FUNCTION_BLOCK StartStopEvents (* Basic Function Block Type *)
  (* Standard: 61499-2 *)
  (* Version 0.0, 18/05/2022, Admin, Schneider Electric, Template *)
  PACKAGE Main;
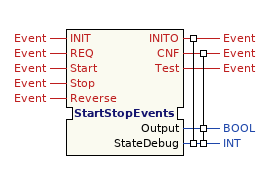
  EVENT_INPUT
    INIT; (* Initialization Request *)
    REQ; (* Normal Execution Request *)
    Start;
    Stop;
    Reverse;
  END_EVENT
  EVENT_OUTPUT
    INITO WITH StateDebug; (* Initialization Confirm *)
    CNF WITH Output, StateDebug; (* Execution Confirmation *)
    Test;
  END_EVENT
  VAR_OUTPUT
    Output : BOOL := FALSE; (* Output event qualifier *)
    StateDebug : INT := -99;
  END_VAR
  VAR
    InternalState : BOOL;
  END_VAR
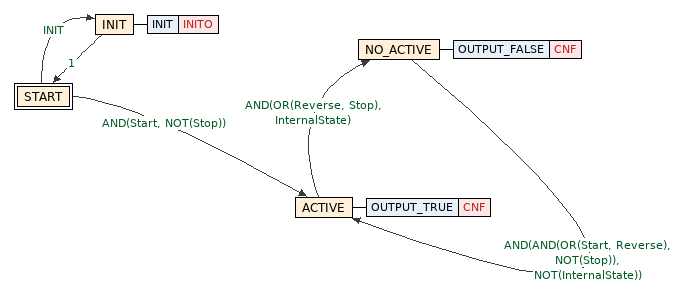
  EC_STATES
    START; (* Initial State *)
    INIT : INIT -> INITO; (* Initialization *)
    ACTIVE : OUTPUT_TRUE -> CNF; (* Normal execution *)
    NO_ACTIVE : OUTPUT_FALSE -> CNF;
  END_STATES
  EC_TRANSITIONS
    START TO INIT := INIT;
    INIT TO START := 1;
    START TO ACTIVE := AND(Start, NOT(Stop));
    ACTIVE TO NO_ACTIVE := AND(OR(Reverse, Stop), InternalState);
    NO_ACTIVE TO ACTIVE := AND(AND(OR(Start, Reverse), NOT(Stop)), NOT(InternalState));
  END_TRANSITIONS
  ALGORITHM INIT IN ST: (* Initialization algorithm *)
;

StateDebug := -10;
  END_ALGORITHM
  ALGORITHM OUTPUT_TRUE IN ST: (* Normally executed algorithm *)
;

Output := TRUE;
InternalState := TRUE;
StateDebug := 1;
Reverse := FALSE;
  END_ALGORITHM
  ALGORITHM OUTPUT_FALSE IN ST:
;

Output := FALSE;
InternalState := FALSE;
StateDebug := -1;
Reverse := FALSE;
  END_ALGORITHM
END_FUNCTION_BLOCK
